// TIA Portal V17 export
// export: Created 2025-07-01T09:58:40.6869858Z, ExportSetting WithDefaults, DisplayName Totally Integrated Automation Portal, DisplayVersion V17 Update 8, DisplayName TIA Portal Openness, DisplayVersion V17 Update 8, DisplayName TIA Portal Version Control Interface, DisplayVersion V17, DisplayName SINAMICS Startdrive Advanced, DisplayVersion V17 SP2, DisplayName SINAMICS Startdrive G110M, G120, G120C, G120D, G120P, G115D, DisplayVersion V17 SP2, DisplayName SINAMICS Startdrive G130, G150, S120, S150, SINAMICS MV, S210, DisplayVersion V17 SP2, DisplayName STEP 7 Professional, DisplayVersion V17 Update 8, DisplayName SINUMERIK ONE STEP 7 Toolbox, DisplayVersion V17 Update 12, DisplayName SINUMERIK ONE PLC Basic Program Plus, DisplayVersion V17 Update 12, DisplayName SINUMERIK 840D sl STEP 7 Toolbox, DisplayVersion V17 Update 12, DisplayName STEP 7 Safety, DisplayVersion V17 Update 6, DisplayName WinCC Advanced, DisplayVersion V17 Update 8
FUNCTION "FC328_CHANNEL_8" : Void   // FC328, LAD
{ S7_Optimized_Access := 'FALSE' }
AUTHOR : ETXETAR
VERSION : 1.0
// stored: AutoNumber false, IsIECCheckEnabled false, SetENOAutomatically false, UDAEnableTagReadback false
   VAR_TEMP
      NC_RESET_CH4 : Bool;
      NC_START_CH4 : Bool;
      MODE_GROUP_1 : Struct
         CHAN_MODE_GROUP : Int;
         ENABLE_OVERRIDE_MP_HT10 : Bool;
         CHAN_OVERRIDE_VALUE : Byte;
         BA3_SOFT_KEY_STOP : Bool;
         MACHINE_IS_ALARM : Bool;
         MACHINE_IS_WARNING : Bool;
         CH_MACHINE_RESET : Bool;
         MPP_PUSH_BUTTON_START : Bool;
         MPP_PUSH_BUTTON_NC_START : Bool;
         MPP_BUTTON_HOME_POS : Bool;
         SEQ_RUNNING : Bool;
      END_STRUCT;
      MODE_GROUP_2 : Struct
         CHAN_MODE_GROUP : Int;
         ENABLE_OVERRIDE_MP_HT10 : Bool;
         CHAN_OVERRIDE_VALUE : Byte;
         BA3_SOFT_KEY_STOP : Bool;
         MACHINE_IS_ALARM : Bool;
         MACHINE_IS_WARNING : Bool;
         CH_MACHINE_RESET : Bool;
         MPP_PUSH_BUTTON_START : Bool;
         MPP_PUSH_BUTTON_NC_START : Bool;
         MPP_BUTTON_HOME_POS : Bool;
         SEQ_RUNNING : Bool;
      END_STRUCT;
      MODE_GROUP_SELECTED : Struct
         CHAN_MODE_GROUP : Int;
         ENABLE_OVERRIDE_MP_HT10 : Bool;
         CHAN_OVERRIDE_VALUE : Byte;
         BA3_SOFT_KEY_STOP : Bool;
         MACHINE_IS_ALARM : Bool;
         MACHINE_IS_WARNING : Bool;
         CH_MACHINE_RESET : Bool;
         MPP_PUSH_BUTTON_START : Bool;
         MPP_PUSH_BUTTON_NC_START : Bool;
         MPP_BUTTON_HOME_POS : Bool;
         SEQ_RUNNING : Bool;
      END_STRUCT;
   END_VAR
   VAR_TEMP   // added for the SCL form of the ladder/FBD networks
      _w1 : Bool;
   END_VAR
BEGIN

REGION Network 1: RESET CHANNEL
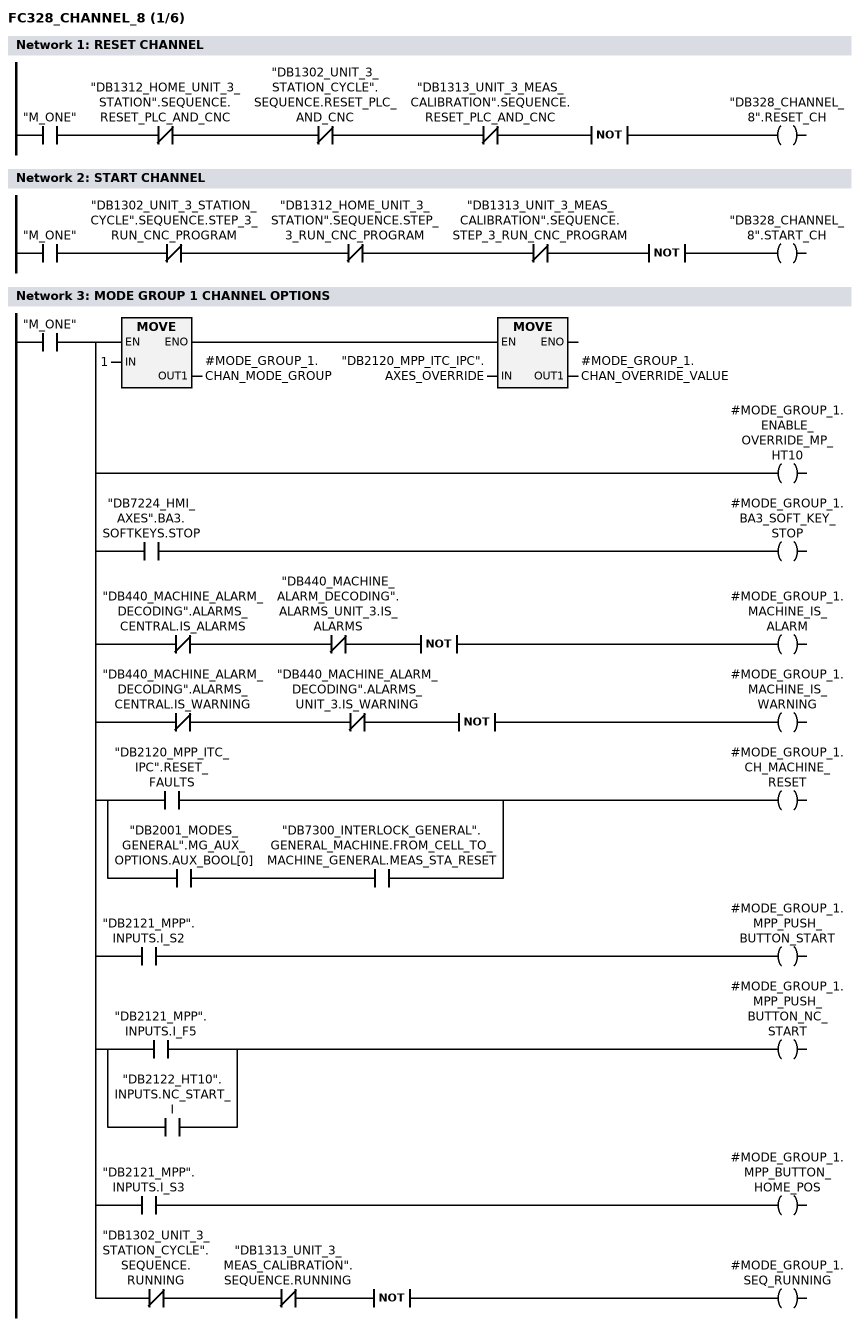
   RUNG wire#powerrail
      Contact( "M_ONE" )
      I_Contact( "DB1312_HOME_UNIT_3_STATION".SEQUENCE.RESET_PLC_AND_CNC )
      I_Contact( "DB1302_UNIT_3_STATION_CYCLE".SEQUENCE.RESET_PLC_AND_CNC )
      I_Contact( "DB1313_UNIT_3_MEAS_CALIBRATION".SEQUENCE.RESET_PLC_AND_CNC )
      Not()
      Coil( "DB328_CHANNEL_8".RESET_CH )
   END_RUNG
   // the same network as SCL:
   "DB328_CHANNEL_8".RESET_CH := NOT ("M_ONE" AND NOT "DB1312_HOME_UNIT_3_STATION".SEQUENCE.RESET_PLC_AND_CNC AND NOT "DB1302_UNIT_3_STATION_CYCLE".SEQUENCE.RESET_PLC_AND_CNC AND NOT "DB1313_UNIT_3_MEAS_CALIBRATION".SEQUENCE.RESET_PLC_AND_CNC);
END_REGION

REGION Network 2: START CHANNEL
   RUNG wire#powerrail
      Contact( "M_ONE" )
      I_Contact( "DB1302_UNIT_3_STATION_CYCLE".SEQUENCE.STEP_3_RUN_CNC_PROGRAM )
      I_Contact( "DB1312_HOME_UNIT_3_STATION".SEQUENCE.STEP_3_RUN_CNC_PROGRAM )
      I_Contact( "DB1313_UNIT_3_MEAS_CALIBRATION".SEQUENCE.STEP_3_RUN_CNC_PROGRAM )
      Not()
      Coil( "DB328_CHANNEL_8".START_CH )
   END_RUNG
   // the same network as SCL:
   "DB328_CHANNEL_8".START_CH := NOT ("M_ONE" AND NOT "DB1302_UNIT_3_STATION_CYCLE".SEQUENCE.STEP_3_RUN_CNC_PROGRAM AND NOT "DB1312_HOME_UNIT_3_STATION".SEQUENCE.STEP_3_RUN_CNC_PROGRAM AND NOT "DB1313_UNIT_3_MEAS_CALIBRATION".SEQUENCE.STEP_3_RUN_CNC_PROGRAM);
END_REGION

REGION Network 3: MODE GROUP 1 CHANNEL OPTIONS
   RUNG wire#powerrail
      Contact( "M_ONE" )
      wire#w1
      Move(in := 1, out1 => #MODE_GROUP_1.CHAN_MODE_GROUP)
      Move(in := "DB2120_MPP_ITC_IPC".AXES_OVERRIDE, out1 => #MODE_GROUP_1.CHAN_OVERRIDE_VALUE)
   END_RUNG
   RUNG wire#w1
      Coil( #MODE_GROUP_1.ENABLE_OVERRIDE_MP_HT10 )
   END_RUNG
   RUNG wire#w1
      Contact( "DB7224_HMI_AXES".BA3.SOFTKEYS.STOP )
      Coil( #MODE_GROUP_1.BA3_SOFT_KEY_STOP )
   END_RUNG
   RUNG wire#w1
      I_Contact( "DB440_MACHINE_ALARM_DECODING".ALARMS_CENTRAL.IS_ALARMS )
      I_Contact( "DB440_MACHINE_ALARM_DECODING".ALARMS_UNIT_3.IS_ALARMS )
      Not()
      Coil( #MODE_GROUP_1.MACHINE_IS_ALARM )
   END_RUNG
   RUNG wire#w1
      I_Contact( "DB440_MACHINE_ALARM_DECODING".ALARMS_CENTRAL.IS_WARNING )
      I_Contact( "DB440_MACHINE_ALARM_DECODING".ALARMS_UNIT_3.IS_WARNING )
      Not()
      Coil( #MODE_GROUP_1.MACHINE_IS_WARNING )
   END_RUNG
   RUNG wire#w1
      Contact( "DB2120_MPP_ITC_IPC".RESET_FAULTS )
      wire#w2
      Coil( #MODE_GROUP_1.CH_MACHINE_RESET )
   END_RUNG
   RUNG wire#w1
      Contact( "DB2001_MODES_GENERAL".MG_AUX_OPTIONS.AUX_BOOL[0] )
      Contact( "DB7300_INTERLOCK_GENERAL".GENERAL_MACHINE.FROM_CELL_TO_MACHINE_GENERAL.MEAS_STA_RESET )
   END_RUNG wire#w2
   RUNG wire#w1
      Contact( "DB2121_MPP".INPUTS.I_S2 )
      Coil( #MODE_GROUP_1.MPP_PUSH_BUTTON_START )
   END_RUNG
   RUNG wire#w1
      Contact( "DB2121_MPP".INPUTS.I_F5 )
      wire#w3
      Coil( #MODE_GROUP_1.MPP_PUSH_BUTTON_NC_START )
   END_RUNG
   RUNG wire#w1
      Contact( "DB2122_HT10".INPUTS.NC_START_I )
   END_RUNG wire#w3
   RUNG wire#w1
      Contact( "DB2121_MPP".INPUTS.I_S3 )
      Coil( #MODE_GROUP_1.MPP_BUTTON_HOME_POS )
   END_RUNG
   RUNG wire#w1
      I_Contact( "DB1302_UNIT_3_STATION_CYCLE".SEQUENCE.RUNNING )
      I_Contact( "DB1313_UNIT_3_MEAS_CALIBRATION".SEQUENCE.RUNNING )
      Not()
      Coil( #MODE_GROUP_1.SEQ_RUNNING )
   END_RUNG
   // the same network as SCL:
   IF "M_ONE" THEN
       #MODE_GROUP_1.CHAN_MODE_GROUP := 1;
       #MODE_GROUP_1.CHAN_OVERRIDE_VALUE := "DB2120_MPP_ITC_IPC".AXES_OVERRIDE;
   END_IF;
   #MODE_GROUP_1.ENABLE_OVERRIDE_MP_HT10 := "M_ONE";
   #MODE_GROUP_1.BA3_SOFT_KEY_STOP := "M_ONE" AND "DB7224_HMI_AXES".BA3.SOFTKEYS.STOP;
   #MODE_GROUP_1.MACHINE_IS_ALARM := NOT ("M_ONE" AND NOT "DB440_MACHINE_ALARM_DECODING".ALARMS_CENTRAL.IS_ALARMS AND NOT "DB440_MACHINE_ALARM_DECODING".ALARMS_UNIT_3.IS_ALARMS);
   #MODE_GROUP_1.MACHINE_IS_WARNING := NOT ("M_ONE" AND NOT "DB440_MACHINE_ALARM_DECODING".ALARMS_CENTRAL.IS_WARNING AND NOT "DB440_MACHINE_ALARM_DECODING".ALARMS_UNIT_3.IS_WARNING);
   #MODE_GROUP_1.CH_MACHINE_RESET := "M_ONE" AND ("DB2120_MPP_ITC_IPC".RESET_FAULTS OR ("DB2001_MODES_GENERAL".MG_AUX_OPTIONS.AUX_BOOL[0] AND "DB7300_INTERLOCK_GENERAL".GENERAL_MACHINE.FROM_CELL_TO_MACHINE_GENERAL.MEAS_STA_RESET));
   #MODE_GROUP_1.MPP_PUSH_BUTTON_START := "M_ONE" AND "DB2121_MPP".INPUTS.I_S2;
   #MODE_GROUP_1.MPP_PUSH_BUTTON_NC_START := "M_ONE" AND ("DB2121_MPP".INPUTS.I_F5 OR "DB2122_HT10".INPUTS.NC_START_I);
   #MODE_GROUP_1.MPP_BUTTON_HOME_POS := "M_ONE" AND "DB2121_MPP".INPUTS.I_S3;
   #MODE_GROUP_1.SEQ_RUNNING := NOT ("M_ONE" AND NOT "DB1302_UNIT_3_STATION_CYCLE".SEQUENCE.RUNNING AND NOT "DB1313_UNIT_3_MEAS_CALIBRATION".SEQUENCE.RUNNING);
END_REGION

REGION Network 4: MODE GROUP 2 CHANNEL OPTIONS
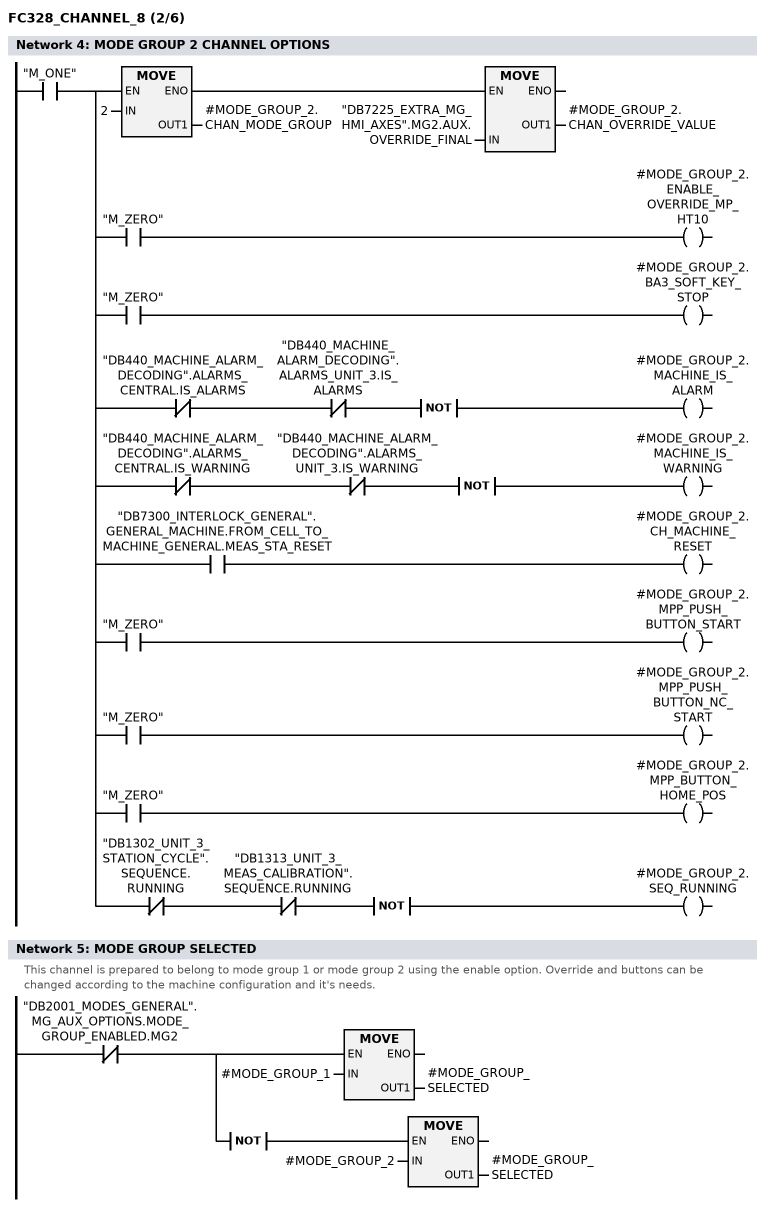
   RUNG wire#powerrail
      Contact( "M_ONE" )
      wire#w1
      Move(in := 2, out1 => #MODE_GROUP_2.CHAN_MODE_GROUP)
      Move(in := "DB7225_EXTRA_MG_HMI_AXES".MG2.AUX.OVERRIDE_FINAL, out1 => #MODE_GROUP_2.CHAN_OVERRIDE_VALUE)
   END_RUNG
   RUNG wire#w1
      Contact( "M_ZERO" )
      Coil( #MODE_GROUP_2.ENABLE_OVERRIDE_MP_HT10 )
   END_RUNG
   RUNG wire#w1
      Contact( "M_ZERO" )
      Coil( #MODE_GROUP_2.BA3_SOFT_KEY_STOP )
   END_RUNG
   RUNG wire#w1
      I_Contact( "DB440_MACHINE_ALARM_DECODING".ALARMS_CENTRAL.IS_ALARMS )
      I_Contact( "DB440_MACHINE_ALARM_DECODING".ALARMS_UNIT_3.IS_ALARMS )
      Not()
      Coil( #MODE_GROUP_2.MACHINE_IS_ALARM )
   END_RUNG
   RUNG wire#w1
      I_Contact( "DB440_MACHINE_ALARM_DECODING".ALARMS_CENTRAL.IS_WARNING )
      I_Contact( "DB440_MACHINE_ALARM_DECODING".ALARMS_UNIT_3.IS_WARNING )
      Not()
      Coil( #MODE_GROUP_2.MACHINE_IS_WARNING )
   END_RUNG
   RUNG wire#w1
      Contact( "DB7300_INTERLOCK_GENERAL".GENERAL_MACHINE.FROM_CELL_TO_MACHINE_GENERAL.MEAS_STA_RESET )
      Coil( #MODE_GROUP_2.CH_MACHINE_RESET )
   END_RUNG
   RUNG wire#w1
      Contact( "M_ZERO" )
      Coil( #MODE_GROUP_2.MPP_PUSH_BUTTON_START )
   END_RUNG
   RUNG wire#w1
      Contact( "M_ZERO" )
      Coil( #MODE_GROUP_2.MPP_PUSH_BUTTON_NC_START )
   END_RUNG
   RUNG wire#w1
      Contact( "M_ZERO" )
      Coil( #MODE_GROUP_2.MPP_BUTTON_HOME_POS )
   END_RUNG
   RUNG wire#w1
      I_Contact( "DB1302_UNIT_3_STATION_CYCLE".SEQUENCE.RUNNING )
      I_Contact( "DB1313_UNIT_3_MEAS_CALIBRATION".SEQUENCE.RUNNING )
      Not()
      Coil( #MODE_GROUP_2.SEQ_RUNNING )
   END_RUNG
   // the same network as SCL:
   IF "M_ONE" THEN
       #MODE_GROUP_2.CHAN_MODE_GROUP := 2;
       #MODE_GROUP_2.CHAN_OVERRIDE_VALUE := "DB7225_EXTRA_MG_HMI_AXES".MG2.AUX.OVERRIDE_FINAL;
   END_IF;
   #MODE_GROUP_2.ENABLE_OVERRIDE_MP_HT10 := "M_ONE" AND "M_ZERO";
   #MODE_GROUP_2.BA3_SOFT_KEY_STOP := "M_ONE" AND "M_ZERO";
   #MODE_GROUP_2.MACHINE_IS_ALARM := NOT ("M_ONE" AND NOT "DB440_MACHINE_ALARM_DECODING".ALARMS_CENTRAL.IS_ALARMS AND NOT "DB440_MACHINE_ALARM_DECODING".ALARMS_UNIT_3.IS_ALARMS);
   #MODE_GROUP_2.MACHINE_IS_WARNING := NOT ("M_ONE" AND NOT "DB440_MACHINE_ALARM_DECODING".ALARMS_CENTRAL.IS_WARNING AND NOT "DB440_MACHINE_ALARM_DECODING".ALARMS_UNIT_3.IS_WARNING);
   #MODE_GROUP_2.CH_MACHINE_RESET := "M_ONE" AND "DB7300_INTERLOCK_GENERAL".GENERAL_MACHINE.FROM_CELL_TO_MACHINE_GENERAL.MEAS_STA_RESET;
   #MODE_GROUP_2.MPP_PUSH_BUTTON_START := "M_ONE" AND "M_ZERO";
   #MODE_GROUP_2.MPP_PUSH_BUTTON_NC_START := "M_ONE" AND "M_ZERO";
   #MODE_GROUP_2.MPP_BUTTON_HOME_POS := "M_ONE" AND "M_ZERO";
   #MODE_GROUP_2.SEQ_RUNNING := NOT ("M_ONE" AND NOT "DB1302_UNIT_3_STATION_CYCLE".SEQUENCE.RUNNING AND NOT "DB1313_UNIT_3_MEAS_CALIBRATION".SEQUENCE.RUNNING);
END_REGION

REGION Network 5: MODE GROUP SELECTED
   // This channel is prepared to belong to mode group 1 or mode group 2 using the enable option. Override and buttons can be changed according to the machine configuration and it's needs.
   RUNG wire#powerrail
      I_Contact( "DB2001_MODES_GENERAL".MG_AUX_OPTIONS.MODE_GROUP_ENABLED.MG2 )
      wire#w1
      Move(in := #MODE_GROUP_1, out1 => #MODE_GROUP_SELECTED)
   END_RUNG
   RUNG wire#w1
      Not()
      Move(in := #MODE_GROUP_2, out1 => #MODE_GROUP_SELECTED)
   END_RUNG
   // the same network as SCL:
   #_w1 := NOT "DB2001_MODES_GENERAL".MG_AUX_OPTIONS.MODE_GROUP_ENABLED.MG2;
   IF #_w1 THEN #MODE_GROUP_SELECTED := #MODE_GROUP_1; END_IF;
   IF NOT #_w1 THEN #MODE_GROUP_SELECTED := #MODE_GROUP_2; END_IF;
END_REGION

REGION Network 6: CALL FB321 CHANNEL 8 / CHANNEL 4 XFLEX-DUO
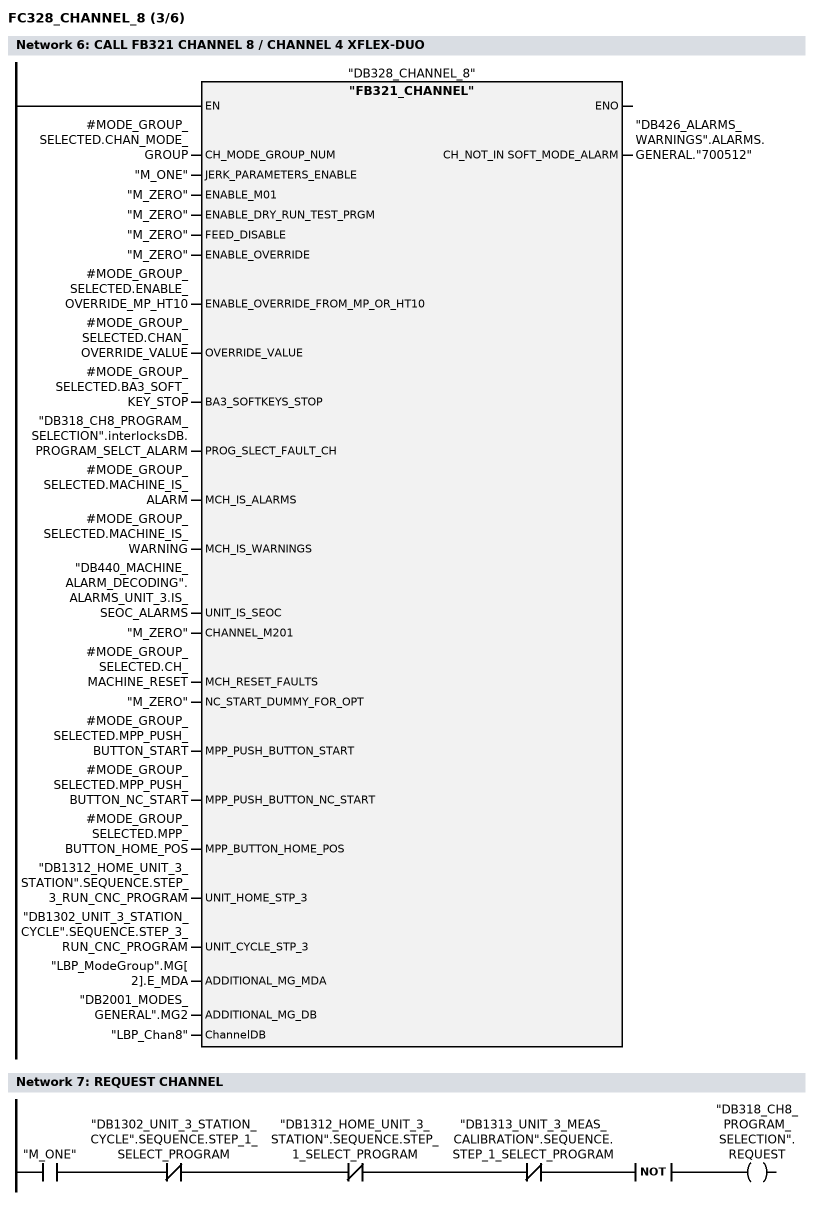
   RUNG wire#powerrail
      "DB328_CHANNEL_8"(CH_MODE_GROUP_NUM := #MODE_GROUP_SELECTED.CHAN_MODE_GROUP, JERK_PARAMETERS_ENABLE := "M_ONE", ENABLE_M01 := "M_ZERO", ENABLE_DRY_RUN_TEST_PRGM := "M_ZERO", FEED_DISABLE := "M_ZERO", ENABLE_OVERRIDE := "M_ZERO", ENABLE_OVERRIDE_FROM_MP_OR_HT10 := #MODE_GROUP_SELECTED.ENABLE_OVERRIDE_MP_HT10, OVERRIDE_VALUE := #MODE_GROUP_SELECTED.CHAN_OVERRIDE_VALUE, BA3_SOFTKEYS_STOP := #MODE_GROUP_SELECTED.BA3_SOFT_KEY_STOP, PROG_SLECT_FAULT_CH := "DB318_CH8_PROGRAM_SELECTION".interlocksDB.PROGRAM_SELCT_ALARM, MCH_IS_ALARMS := #MODE_GROUP_SELECTED.MACHINE_IS_ALARM, MCH_IS_WARNINGS := #MODE_GROUP_SELECTED.MACHINE_IS_WARNING, UNIT_IS_SEOC := "DB440_MACHINE_ALARM_DECODING".ALARMS_UNIT_3.IS_SEOC_ALARMS, CHANNEL_M201 := "M_ZERO", MCH_RESET_FAULTS := #MODE_GROUP_SELECTED.CH_MACHINE_RESET, NC_START_DUMMY_FOR_OPT := "M_ZERO", MPP_PUSH_BUTTON_START := #MODE_GROUP_SELECTED.MPP_PUSH_BUTTON_START, MPP_PUSH_BUTTON_NC_START := #MODE_GROUP_SELECTED.MPP_PUSH_BUTTON_NC_START, MPP_BUTTON_HOME_POS := #MODE_GROUP_SELECTED.MPP_BUTTON_HOME_POS, UNIT_HOME_STP_3 := "DB1312_HOME_UNIT_3_STATION".SEQUENCE.STEP_3_RUN_CNC_PROGRAM, UNIT_CYCLE_STP_3 := "DB1302_UNIT_3_STATION_CYCLE".SEQUENCE.STEP_3_RUN_CNC_PROGRAM, ADDITIONAL_MG_MDA := "LBP_ModeGroup".MG[2].E_MDA, ADDITIONAL_MG_DB := "DB2001_MODES_GENERAL".MG2, ChannelDB := "LBP_Chan8", "CH_NOT_IN SOFT_MODE_ALARM" => "DB426_ALARMS_WARNINGS".ALARMS.GENERAL."700512")
   END_RUNG
   // the same network as SCL:
   "DB328_CHANNEL_8"(CH_MODE_GROUP_NUM := #MODE_GROUP_SELECTED.CHAN_MODE_GROUP,   // "FB321_CHANNEL"
                     JERK_PARAMETERS_ENABLE := "M_ONE",
                     ENABLE_M01 := "M_ZERO",
                     ENABLE_DRY_RUN_TEST_PRGM := "M_ZERO",
                     FEED_DISABLE := "M_ZERO",
                     ENABLE_OVERRIDE := "M_ZERO",
                     ENABLE_OVERRIDE_FROM_MP_OR_HT10 := #MODE_GROUP_SELECTED.ENABLE_OVERRIDE_MP_HT10,
                     OVERRIDE_VALUE := #MODE_GROUP_SELECTED.CHAN_OVERRIDE_VALUE,
                     BA3_SOFTKEYS_STOP := #MODE_GROUP_SELECTED.BA3_SOFT_KEY_STOP,
                     PROG_SLECT_FAULT_CH := "DB318_CH8_PROGRAM_SELECTION".interlocksDB.PROGRAM_SELCT_ALARM,
                     MCH_IS_ALARMS := #MODE_GROUP_SELECTED.MACHINE_IS_ALARM,
                     MCH_IS_WARNINGS := #MODE_GROUP_SELECTED.MACHINE_IS_WARNING,
                     UNIT_IS_SEOC := "DB440_MACHINE_ALARM_DECODING".ALARMS_UNIT_3.IS_SEOC_ALARMS,
                     CHANNEL_M201 := "M_ZERO",
                     MCH_RESET_FAULTS := #MODE_GROUP_SELECTED.CH_MACHINE_RESET,
                     NC_START_DUMMY_FOR_OPT := "M_ZERO",
                     MPP_PUSH_BUTTON_START := #MODE_GROUP_SELECTED.MPP_PUSH_BUTTON_START,
                     MPP_PUSH_BUTTON_NC_START := #MODE_GROUP_SELECTED.MPP_PUSH_BUTTON_NC_START,
                     MPP_BUTTON_HOME_POS := #MODE_GROUP_SELECTED.MPP_BUTTON_HOME_POS,
                     UNIT_HOME_STP_3 := "DB1312_HOME_UNIT_3_STATION".SEQUENCE.STEP_3_RUN_CNC_PROGRAM,
                     UNIT_CYCLE_STP_3 := "DB1302_UNIT_3_STATION_CYCLE".SEQUENCE.STEP_3_RUN_CNC_PROGRAM,
                     ADDITIONAL_MG_MDA := "LBP_ModeGroup".MG[2].E_MDA,
                     ADDITIONAL_MG_DB := "DB2001_MODES_GENERAL".MG2,
                     ChannelDB := "LBP_Chan8",
                     "CH_NOT_IN SOFT_MODE_ALARM" => "DB426_ALARMS_WARNINGS".ALARMS.GENERAL."700512");
END_REGION

REGION Network 7: REQUEST CHANNEL
   RUNG wire#powerrail
      Contact( "M_ONE" )
      I_Contact( "DB1302_UNIT_3_STATION_CYCLE".SEQUENCE.STEP_1_SELECT_PROGRAM )
      I_Contact( "DB1312_HOME_UNIT_3_STATION".SEQUENCE.STEP_1_SELECT_PROGRAM )
      I_Contact( "DB1313_UNIT_3_MEAS_CALIBRATION".SEQUENCE.STEP_1_SELECT_PROGRAM )
      Not()
      Coil( "DB318_CH8_PROGRAM_SELECTION".REQUEST )
   END_RUNG
   // the same network as SCL:
   "DB318_CH8_PROGRAM_SELECTION".REQUEST := NOT ("M_ONE" AND NOT "DB1302_UNIT_3_STATION_CYCLE".SEQUENCE.STEP_1_SELECT_PROGRAM AND NOT "DB1312_HOME_UNIT_3_STATION".SEQUENCE.STEP_1_SELECT_PROGRAM AND NOT "DB1313_UNIT_3_MEAS_CALIBRATION".SEQUENCE.STEP_1_SELECT_PROGRAM);
END_REGION

REGION Network 8: CALL FB311 CHANNEL PROGRAM SELECTION / CHANNEL 4 X-FLEX DUO
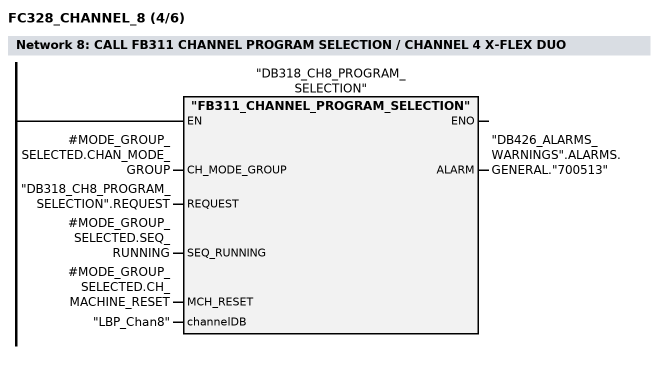
   RUNG wire#powerrail
      "DB318_CH8_PROGRAM_SELECTION"(CH_MODE_GROUP := #MODE_GROUP_SELECTED.CHAN_MODE_GROUP, REQUEST := "DB318_CH8_PROGRAM_SELECTION".REQUEST, SEQ_RUNNING := #MODE_GROUP_SELECTED.SEQ_RUNNING, MCH_RESET := #MODE_GROUP_SELECTED.CH_MACHINE_RESET, channelDB := "LBP_Chan8", ALARM => "DB426_ALARMS_WARNINGS".ALARMS.GENERAL."700513")
   END_RUNG
   // the same network as SCL:
   "DB318_CH8_PROGRAM_SELECTION"(CH_MODE_GROUP := #MODE_GROUP_SELECTED.CHAN_MODE_GROUP,   // "FB311_CHANNEL_PROGRAM_SELECTION"
                           REQUEST := "DB318_CH8_PROGRAM_SELECTION".REQUEST,
                           SEQ_RUNNING := #MODE_GROUP_SELECTED.SEQ_RUNNING,
                           MCH_RESET := #MODE_GROUP_SELECTED.CH_MACHINE_RESET,
                           channelDB := "LBP_Chan8",
                           ALARM => "DB426_ALARMS_WARNINGS".ALARMS.GENERAL."700513");
END_REGION

REGION Network 9: CALL FB301 CHANNEL READ AXES POSITIONS
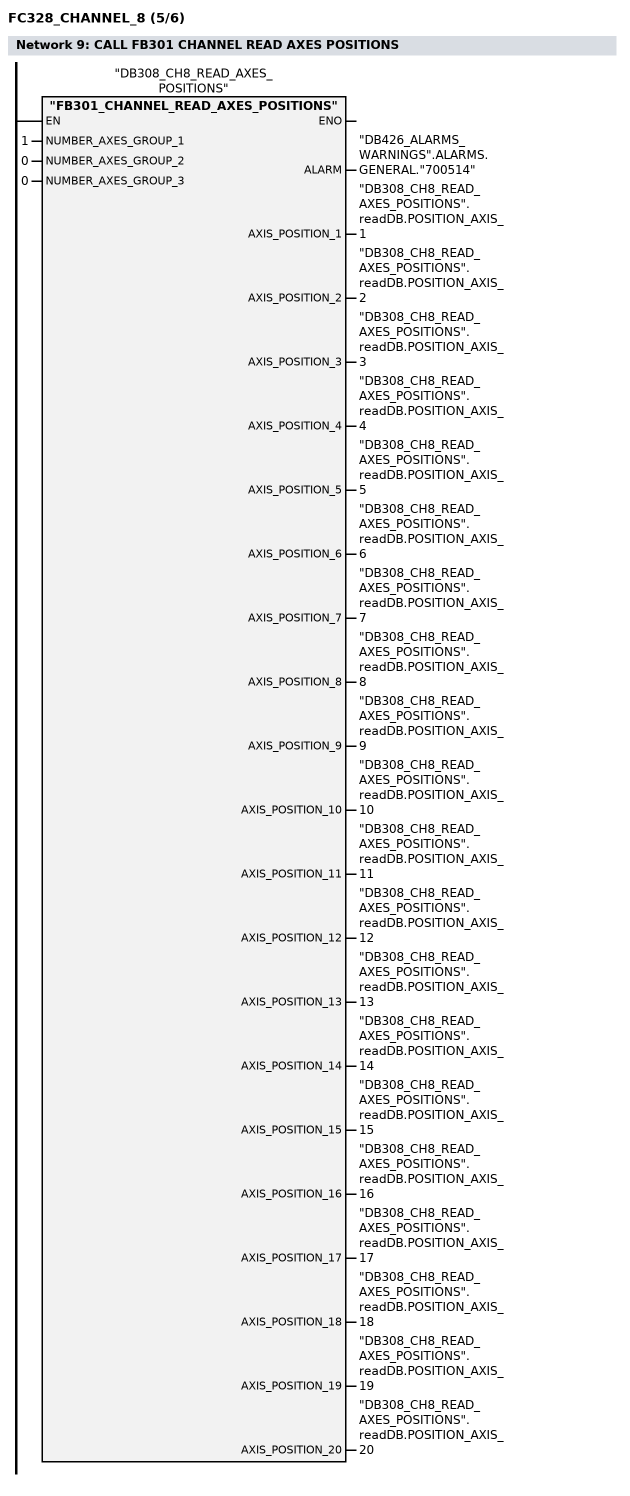
   RUNG wire#powerrail
      "DB308_CH8_READ_AXES_POSITIONS"(NUMBER_AXES_GROUP_1 := 1, NUMBER_AXES_GROUP_2 := 0, NUMBER_AXES_GROUP_3 := 0, ALARM => "DB426_ALARMS_WARNINGS".ALARMS.GENERAL."700514", AXIS_POSITION_1 => "DB308_CH8_READ_AXES_POSITIONS".readDB.POSITION_AXIS_1, AXIS_POSITION_2 => "DB308_CH8_READ_AXES_POSITIONS".readDB.POSITION_AXIS_2, AXIS_POSITION_3 => "DB308_CH8_READ_AXES_POSITIONS".readDB.POSITION_AXIS_3, AXIS_POSITION_4 => "DB308_CH8_READ_AXES_POSITIONS".readDB.POSITION_AXIS_4, AXIS_POSITION_5 => "DB308_CH8_READ_AXES_POSITIONS".readDB.POSITION_AXIS_5, AXIS_POSITION_6 => "DB308_CH8_READ_AXES_POSITIONS".readDB.POSITION_AXIS_6, AXIS_POSITION_7 => "DB308_CH8_READ_AXES_POSITIONS".readDB.POSITION_AXIS_7, AXIS_POSITION_8 => "DB308_CH8_READ_AXES_POSITIONS".readDB.POSITION_AXIS_8, AXIS_POSITION_9 => "DB308_CH8_READ_AXES_POSITIONS".readDB.POSITION_AXIS_9, AXIS_POSITION_10 => "DB308_CH8_READ_AXES_POSITIONS".readDB.POSITION_AXIS_10, AXIS_POSITION_11 => "DB308_CH8_READ_AXES_POSITIONS".readDB.POSITION_AXIS_11, AXIS_POSITION_12 => "DB308_CH8_READ_AXES_POSITIONS".readDB.POSITION_AXIS_12, AXIS_POSITION_13 => "DB308_CH8_READ_AXES_POSITIONS".readDB.POSITION_AXIS_13, AXIS_POSITION_14 => "DB308_CH8_READ_AXES_POSITIONS".readDB.POSITION_AXIS_14, AXIS_POSITION_15 => "DB308_CH8_READ_AXES_POSITIONS".readDB.POSITION_AXIS_15, AXIS_POSITION_16 => "DB308_CH8_READ_AXES_POSITIONS".readDB.POSITION_AXIS_16, AXIS_POSITION_17 => "DB308_CH8_READ_AXES_POSITIONS".readDB.POSITION_AXIS_17, AXIS_POSITION_18 => "DB308_CH8_READ_AXES_POSITIONS".readDB.POSITION_AXIS_18, AXIS_POSITION_19 => "DB308_CH8_READ_AXES_POSITIONS".readDB.POSITION_AXIS_19, AXIS_POSITION_20 => "DB308_CH8_READ_AXES_POSITIONS".readDB.POSITION_AXIS_20)
   END_RUNG
   // the same network as SCL:
   "DB308_CH8_READ_AXES_POSITIONS"(NUMBER_AXES_GROUP_1 := 1,   // "FB301_CHANNEL_READ_AXES_POSITIONS"
                           NUMBER_AXES_GROUP_2 := 0,
                           NUMBER_AXES_GROUP_3 := 0,
                           ALARM => "DB426_ALARMS_WARNINGS".ALARMS.GENERAL."700514",
                           AXIS_POSITION_1 => "DB308_CH8_READ_AXES_POSITIONS".readDB.POSITION_AXIS_1,
                           AXIS_POSITION_2 => "DB308_CH8_READ_AXES_POSITIONS".readDB.POSITION_AXIS_2,
                           AXIS_POSITION_3 => "DB308_CH8_READ_AXES_POSITIONS".readDB.POSITION_AXIS_3,
                           AXIS_POSITION_4 => "DB308_CH8_READ_AXES_POSITIONS".readDB.POSITION_AXIS_4,
                           AXIS_POSITION_5 => "DB308_CH8_READ_AXES_POSITIONS".readDB.POSITION_AXIS_5,
                           AXIS_POSITION_6 => "DB308_CH8_READ_AXES_POSITIONS".readDB.POSITION_AXIS_6,
                           AXIS_POSITION_7 => "DB308_CH8_READ_AXES_POSITIONS".readDB.POSITION_AXIS_7,
                           AXIS_POSITION_8 => "DB308_CH8_READ_AXES_POSITIONS".readDB.POSITION_AXIS_8,
                           AXIS_POSITION_9 => "DB308_CH8_READ_AXES_POSITIONS".readDB.POSITION_AXIS_9,
                           AXIS_POSITION_10 => "DB308_CH8_READ_AXES_POSITIONS".readDB.POSITION_AXIS_10,
                           AXIS_POSITION_11 => "DB308_CH8_READ_AXES_POSITIONS".readDB.POSITION_AXIS_11,
                           AXIS_POSITION_12 => "DB308_CH8_READ_AXES_POSITIONS".readDB.POSITION_AXIS_12,
                           AXIS_POSITION_13 => "DB308_CH8_READ_AXES_POSITIONS".readDB.POSITION_AXIS_13,
                           AXIS_POSITION_14 => "DB308_CH8_READ_AXES_POSITIONS".readDB.POSITION_AXIS_14,
                           AXIS_POSITION_15 => "DB308_CH8_READ_AXES_POSITIONS".readDB.POSITION_AXIS_15,
                           AXIS_POSITION_16 => "DB308_CH8_READ_AXES_POSITIONS".readDB.POSITION_AXIS_16,
                           AXIS_POSITION_17 => "DB308_CH8_READ_AXES_POSITIONS".readDB.POSITION_AXIS_17,
                           AXIS_POSITION_18 => "DB308_CH8_READ_AXES_POSITIONS".readDB.POSITION_AXIS_18,
                           AXIS_POSITION_19 => "DB308_CH8_READ_AXES_POSITIONS".readDB.POSITION_AXIS_19,
                           AXIS_POSITION_20 => "DB308_CH8_READ_AXES_POSITIONS".readDB.POSITION_AXIS_20);
END_REGION

REGION Network 10: CALL FC353 NCK M UNIT 03 / CALL FC1182
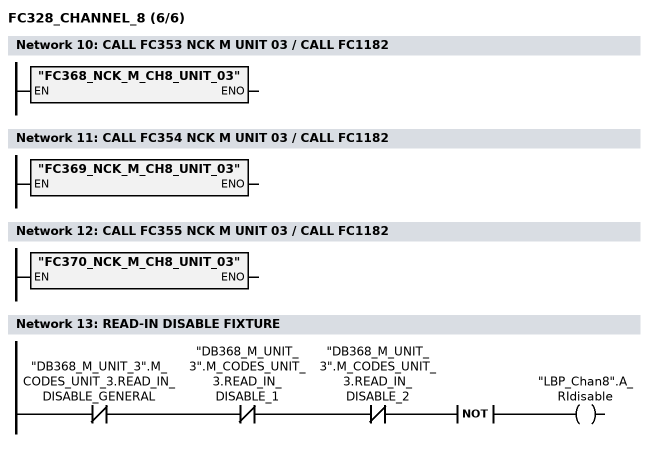
   RUNG wire#powerrail
      "FC368_NCK_M_CH8_UNIT_03"()
   END_RUNG
   // the same network as SCL:
   "FC368_NCK_M_CH8_UNIT_03"();
END_REGION

REGION Network 11: CALL FC354 NCK M UNIT 03 / CALL FC1182
   RUNG wire#powerrail
      "FC369_NCK_M_CH8_UNIT_03"()
   END_RUNG
   // the same network as SCL:
   "FC369_NCK_M_CH8_UNIT_03"();
END_REGION

REGION Network 12: CALL FC355 NCK M UNIT 03 / CALL FC1182
   RUNG wire#powerrail
      "FC370_NCK_M_CH8_UNIT_03"()
   END_RUNG
   // the same network as SCL:
   "FC370_NCK_M_CH8_UNIT_03"();
END_REGION

REGION Network 13: READ-IN DISABLE FIXTURE
   RUNG wire#powerrail
      I_Contact( "DB368_M_UNIT_3".M_CODES_UNIT_3.READ_IN_DISABLE_GENERAL )
      I_Contact( "DB368_M_UNIT_3".M_CODES_UNIT_3.READ_IN_DISABLE_1 )
      I_Contact( "DB368_M_UNIT_3".M_CODES_UNIT_3.READ_IN_DISABLE_2 )
      Not()
      Coil( "LBP_Chan8".A_RIdisable )
   END_RUNG
   // the same network as SCL:
   "LBP_Chan8".A_RIdisable := NOT (NOT "DB368_M_UNIT_3".M_CODES_UNIT_3.READ_IN_DISABLE_GENERAL AND NOT "DB368_M_UNIT_3".M_CODES_UNIT_3.READ_IN_DISABLE_1 AND NOT "DB368_M_UNIT_3".M_CODES_UNIT_3.READ_IN_DISABLE_2);
END_REGION
END_FUNCTION
